PROGRAM RETURN_LASER
VAR_INPUT

END_VAR

VAR
	TMR_DELAY: TON;
	TMR_DELAY1: TON;
	TMR_DELAY2: TON;
END_VAR

CASE SORTER_VAR.I_CASE OF
0: //standby near lotbox
	IF SORTER_VAR.ACTIVE_ID=6 THEN
		SORTER_VAR.ACTIVE_ID:=1;
	END_IF

	CASE SORTER_VAR.I_CURRENT_TRANSACTION.TRANSPORT_INDEX OF
		2 : 
			SORTER_VAR.O_STOPPER_TRANSFER_B:=FALSE;			
			LASER_MOVE(STEP_DATA_1:=0,//3,
				STEP_DATA_2:=1,
				STEP_DATA_3:=12,
				STEP_DATA_4:=0,
				STEP_DATA_5:=1);
		1 : 
			SORTER_VAR.O_STOPPER_TRANSFER_A:=FALSE;
			LASER_MOVE(STEP_DATA_1:=0,//3,
				STEP_DATA_2:=1,
				STEP_DATA_3:=12,
				STEP_DATA_4:=1,
				STEP_DATA_5:=0);
	END_CASE			
	SORTER_VAR.O_VACUUM_On:=FALSE;
	SORTER_VAR.O_VACUUM_OFF:=FALSE;	
	TMR_DELAY(IN:=FALSE);

1://ready for picking up
	IF SORTER_VAR.ACTIVE_ID=6 THEN
		SORTER_VAR.ACTIVE_ID:=1;
	END_IF

		CASE SORTER_VAR.I_CURRENT_TRANSACTION.TRANSPORT_INDEX OF
		1:
			SORTER_VAR.I_RETURN_DONE_A:=FALSE;
		
		2:
			SORTER_VAR.I_RETURN_DONE_B:=FALSE;
	END_CASE
	LASER_MOVE(STEP_DATA_1:=0,
				STEP_DATA_2:=1,
				STEP_DATA_3:=11,
				STEP_DATA_4:=0,
				STEP_DATA_5:=0);	
			
2://ready for picking up
	IF SORTER_VAR.ACTIVE_ID=6 THEN
		SORTER_VAR.ACTIVE_ID:=1;
	END_IF
	TMR_DELAY(IN:=TRUE,PT:=T#1S);
	IF TMR_DELAY.Q THEN
	CASE SORTER_VAR.I_CURRENT_TRANSACTION.TRANSPORT_INDEX OF
	1:		
		//IF SORTER_VAR.I_LASER_TRANSFER_AT_BACK_A THEN
		LASER_MOVE(STEP_DATA_1:=SORTER_VAR.I_CURRENT_TRANSACTION.TRANSPORT_INDEX+5,
				STEP_DATA_2:=1,
				STEP_DATA_3:=11,
				STEP_DATA_4:=0,
				STEP_DATA_5:=0);
		//END_IF
	2:
		//IF SORTER_VAR.I_LASER_TRANSFER_AT_BACK_B THEN
		LASER_MOVE(STEP_DATA_1:=SORTER_VAR.I_CURRENT_TRANSACTION.TRANSPORT_INDEX+5,
				STEP_DATA_2:=1,
				STEP_DATA_3:=11,
				STEP_DATA_4:=0,
				STEP_DATA_5:=0);
	//END_IF
	END_CASE
	END_IF
		
3://VACUUM AND TAKEUP
	IF SORTER_VAR.ACTIVE_ID=6 THEN
		SORTER_VAR.ACTIVE_ID:=1;
	END_IF

	LASER_MOVE(STEP_DATA_1:=SORTER_VAR.I_CURRENT_TRANSACTION.TRANSPORT_INDEX+5,
				STEP_DATA_2:=5,
				STEP_DATA_3:=11,
				STEP_DATA_4:=0,
				STEP_DATA_5:=0);
	SORTER_VAR.O_VACUUM_On:=TRUE;
	SORTER_VAR.O_VACUUM_OFF:=FALSE;
	
4://MOVE BACK 10MM
	IF SORTER_VAR.ACTIVE_ID=6 THEN
		SORTER_VAR.ACTIVE_ID:=1;
	END_IF
	
	LASER_MOVE(STEP_DATA_1:=SORTER_VAR.I_CURRENT_TRANSACTION.TRANSPORT_INDEX+5,
				STEP_DATA_2:=1,
				STEP_DATA_3:=12,
				STEP_DATA_4:=0,
				STEP_DATA_5:=0);

5://MOVE UP 16MM
	IF SORTER_VAR.ACTIVE_ID=6 THEN
		SORTER_VAR.ACTIVE_ID:=1;
	END_IF
	LASER_MOVE(STEP_DATA_1:=SORTER_VAR.I_CURRENT_TRANSACTION.TRANSPORT_INDEX+5,
				STEP_DATA_2:=1,
				STEP_DATA_3:=SORTER_VAR.I_CURRENT_TRANSACTION.JIG_INDEX_RETURN,
				STEP_DATA_4:=0,
				STEP_DATA_5:=0);
	(*
	IF NOT SORTER_VAR.I_VACUUM_On THEN
		LASER_MOVE(STEP_DATA_1:=SORTER_VAR.I_CURRENT_TRANSACTION.TRANSPORT_INDEX+5,
				STEP_DATA_2:=2,
				STEP_DATA_3:=12,
				STEP_DATA_4:=0,
				STEP_DATA_5:=0);
	ELSE
		SORTER_VAR.O_VACUUM_On:=TRUE;
		SORTER_VAR.O_VACUUM_OFF:=FALSE;
	END_IF
	*)
				
6://WAIT THEN MOVE TO NEAR BOX
	IF SORTER_VAR.ACTIVE_ID=6 THEN
		SORTER_VAR.ACTIVE_ID:=1;
	END_IF
	TMR_DELAY1(IN:=TRUE,PT:=T#3S);
	IF TMR_DELAY1.Q THEN
		LASER_MOVE(STEP_DATA_1:=SORTER_VAR.I_CURRENT_TRANSACTION.STATION_NUMBER_RETURN,
				STEP_DATA_2:=2,
				STEP_DATA_3:=14,
				STEP_DATA_4:=0,
				STEP_DATA_5:=0);
	END_IF
	
				
7://vacuum position 
	IF SORTER_VAR.ACTIVE_ID=6 THEN
		SORTER_VAR.ACTIVE_ID:=1;
	END_IF
	SORTER_VAR.I_CASE:=SORTER_VAR.I_CASE+1;
	(*
	TMR_DELAY(IN:=TRUE,PT:=T#1S);
	IF TMR_DELAY.Q THEN
			LASER_MOVE(STEP_DATA_1:=SORTER_VAR.I_CURRENT_TRANSACTION.STATION_NUMBER_RETURN,
				STEP_DATA_2:=2,
				STEP_DATA_3:=14,
				STEP_DATA_4:=0,
				STEP_DATA_5:=0);
	END_IF
		*)		
8://INSERT INTO LOTBOX
	IF SORTER_VAR.ACTIVE_ID=6 THEN
		SORTER_VAR.ACTIVE_ID:=1;
	END_IF
	TMR_DELAY(IN:=FALSE);
	LASER_MOVE(STEP_DATA_1:=SORTER_VAR.I_CURRENT_TRANSACTION.STATION_NUMBER_RETURN,
				STEP_DATA_2:=3,
				STEP_DATA_3:=16,
				STEP_DATA_4:=0,
				STEP_DATA_5:=0);
				
9://MOVE BACK
	IF SORTER_VAR.ACTIVE_ID=6 THEN
		SORTER_VAR.ACTIVE_ID:=1;
	END_IF
	TMR_DELAY2 (IN:=TRUE,PT:=T#2S);
	IF TMR_DELAY2.Q THEN
		LASER_MOVE(STEP_DATA_1:=SORTER_VAR.I_CURRENT_TRANSACTION.STATION_NUMBER_RETURN,
				STEP_DATA_2:=3,
				STEP_DATA_3:=SORTER_VAR.I_CURRENT_TRANSACTION.JIG_INDEX_RETURN,
				STEP_DATA_4:=0,
				STEP_DATA_5:=0);
	END_IF
	SORTER_VAR.O_VACUUM_On:=FALSE;
	SORTER_VAR.O_VACUUM_OFF:=TRUE;
10: //standby near lotbox
	
	IF SORTER_VAR.ACTIVE_ID=6 THEN
		SORTER_VAR.ACTIVE_ID:=1;
	END_IF
LASER_MOVE(STEP_DATA_1:=SORTER_VAR.I_CURRENT_TRANSACTION.STATION_NUMBER_RETURN,
				STEP_DATA_2:=1,
				STEP_DATA_3:=SORTER_VAR.I_CURRENT_TRANSACTION.JIG_INDEX_RETURN,
				STEP_DATA_4:=0,
				STEP_DATA_5:=0);
	(*
	IF SORTER_VAR.I_VACUUM_ON THEN
		LASER_MOVE(STEP_DATA_1:=SORTER_VAR.I_CURRENT_TRANSACTION.STATION_NUMBER_RETURN,
				STEP_DATA_2:=4,
				STEP_DATA_3:=SORTER_VAR.I_CURRENT_TRANSACTION.JIG_INDEX_RETURN,
				STEP_DATA_4:=0,
				STEP_DATA_5:=0);
	ELSE
		SORTER_VAR.O_VACUUM_ON:=FALSE;
		SORTER_VAR.O_VACUUM_OFF:=TRUE;			
	END_IF
	*)
				
11://vacuum position 
	IF SORTER_VAR.ACTIVE_ID=6 THEN
		SORTER_VAR.ACTIVE_ID:=1;
	END_IF
	LASER_MOVE(STEP_DATA_1:=0,
				STEP_DATA_2:=1,
				STEP_DATA_3:=4,
				STEP_DATA_4:=0,
				STEP_DATA_5:=0);
	IF SORTER_VAR.ACTIVE_ID=3 THEN
		SORTER_VAR.O_VACUUM_ON:=FALSE;
		SORTER_VAR.O_VACUUM_OFF:=FALSE;	
	END_IF
	
			
		
100:
	
	SORTER_VAR.O_VACUUM_On:=FALSE;
	SORTER_VAR.O_VACUUM_OFF:=FALSE;
END_CASE 
IF SORTER_VAR.I_CASE=12 THEN
			CASE SORTER_VAR.I_CURRENT_TRANSACTION.TRANSPORT_INDEX OF
		1:
			SORTER_VAR.I_RETURN_DONE_A:=TRUE;
		
		2:
			SORTER_VAR.I_RETURN_DONE_B:=TRUE;
	END_CASE
	IF SORTER_VAR.I_RETURN_DONE_A OR SORTER_VAR.I_RETURN_DONE_B THEN
		FLAG_VAR.ALLOW_EXECUTE_RETURN_LASER:=FALSE;
		TMR_DELAY(IN:=FALSE);
		TMR_DELAY1(IN:=FALSE);
		TMR_DELAY2(IN:=FALSE);
		
		SORTER_VAR.I_CASE:=100;
	END_IF
END_IF

END_PROGRAM

(* stored: Version 1.1.0.1, ProductVersion 3.1.4020.12
   POU RETURN_LASER: Id {1114e93a-06c3-45fb-a632-c3bb59274df1}, SpecialFunc None *)
